Universal Robots PolyScope program: floor corner homing new positions.urp

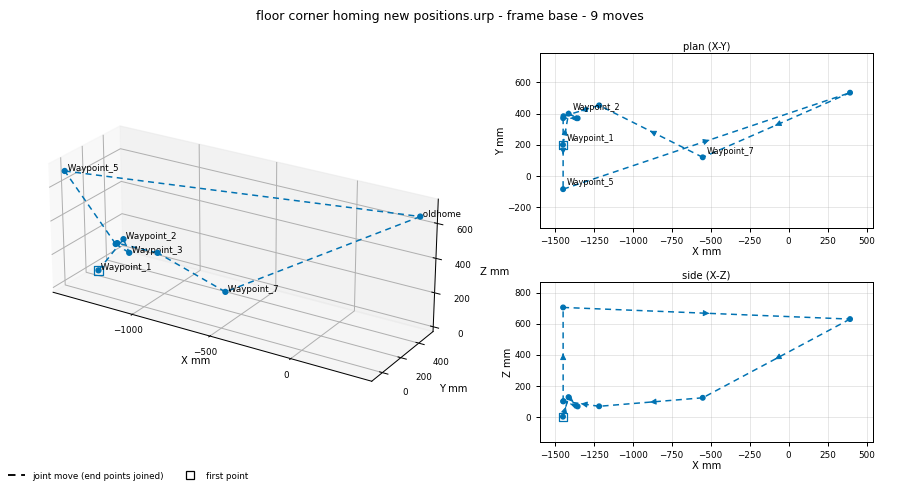
[picture p0: tool path of floor corner homing new positions.urp in frame base, 9 of 9 moves have a stored position in this frame; points joined in program order, loops and branches not executed]
Program floor corner homing new positions (installation=default directory=/programs createdIn=5.21.3 lastSavedIn=5.21.3 robotSerialNumber=20246801938)
Calibrated DH parameters: a=[-0.000071, -0.790281, -0.600694, 0.000061, -0.000039, 0]; d=[0.236272, 604.465945, 132.116513, -736.382239, 0.159268, 0.154005]; alpha=[1.570254, -0.000567, 0.000559, 1.571709, -1.56999, 0]; deltaTheta=[0, -0.409357, 7.293326, -0.600784, -0.000001, -0.000001]
InitVariablesNode
Robot Program (runOnlyOnce=false)
  MoveJ speed 60 deg/s, acceleration 80 deg/s^2 (useActiveTCP=true optimoveEnabled=false optiMoveSpeed=0.3 optiMoveAcceleration=0.09) feature=Base
    Waypoint Waypoint_1: TCP in base x=-1446.032 y=200.324 z=4.429 mm, rx=0.6896 ry=-1.8416 rz=-1.8249 rad; joints [196.593, -160.95, -81.524, 59.369, -337.106, 181.31] deg; TCP offset x=-1.032 y=-18.062 z=285.234 mm, rx=0 ry=0 rz=0 rad
    'left side'
    Waypoint Waypoint_2: TCP in base x=-1410.202 y=399.754 z=129.976 mm, rx=1.3177 ry=-0.7191 rz=-0.5621 rad; joints [156.377, -143.495, -78.511, -125.189, -154.526, 20.301] deg
    'right side'
  MoveJ speed 60 deg/s, acceleration 80 deg/s^2 (useActiveTCP=true optimoveEnabled=false optiMoveSpeed=0.3 optiMoveAcceleration=0.09) feature=Base
    Waypoint Waypoint_3: TCP in base x=-1351.883 y=370.369 z=70.225 mm, rx=1.5108 ry=-0.641 rz=-0.6179 rad; joints [156.251, -143.509, -78.399, -143.327, -157.711, -4.811] deg
    'right side'
    Waypoint Waypoint_4: TCP in base x=-1444.822 y=371.093 z=102.597 mm, rx=0.4492 ry=-1.9864 rz=-2.0242 rad; joints [190.505, -143.519, -77.123, -135.998, -13.155, -5.105] deg
    'left side'
    Waypoint Waypoint_5: TCP in base x=-1445.122 y=-84.303 z=704.854 mm, rx=0.0345 ry=-0.0316 rz=-0.5937 rad; joints [190.517, -143.524, -77.184, -51.731, -90.869, 45.38] deg
    'bottom side'
  'cool so how do we get there'
  MoveJ speed 60 deg/s, acceleration 80 deg/s^2 (useActiveTCP=true optimoveEnabled=false optiMoveSpeed=0.3 optiMoveAcceleration=0.09) feature=Base
    Waypoint oldhome: TCP in base x=394.188 y=534.376 z=630.191 mm, rx=0.0578 ry=2.126 rz=2.1341 rad; joints [-198.279, -117.801, 133.277, -12.745, -11.485, -6.332] deg
    'start from test teach position'
    Waypoint Waypoint_7: TCP in base x=-549.992 y=120.05 z=125.647 mm, rx=1.5708 ry=0 rz=0 rad; joints [-60.367, -57.92, 123.557, -65.577, -60.303, -0.037] deg
    'ttp'
    Waypoint Waypoint_8: TCP in base x=-1214.239 y=453.022 z=71.161 mm, rx=1.2668 ry=-0.8224 rz=-1.0275 rad; joints [-48.516, -43.888, 108.98, -87.586, 22.115, 17.9] deg
    'point they picked'
  MoveJ speed 60 deg/s, acceleration 80 deg/s^2 (useActiveTCP=true optimoveEnabled=false optiMoveSpeed=0.3 optiMoveAcceleration=0.09) feature=Base
    Waypoint Waypoint_6: TCP in base x=-1442.844 y=383.579 z=103.953 mm, rx=0.4388 ry=-1.991 rz=-2.0287 rad; joints [-170, -143.522, -77, -135.998, -13.154, -5.105] deg
    'left side point but base rotated back to normal'
